INTERFACE ITF_CommunicationModul_1

METHOD Connect : BOOL
VAR_INPUT
END_VAR
END_METHOD

PROPERTY Connected : BOOL
GET
END_GET
END_PROPERTY

METHOD Disconnect : BOOL
VAR_INPUT
END_VAR
END_METHOD

METHOD ResetConnection : BOOL
VAR_INPUT
END_VAR
END_METHOD

END_INTERFACE

(* stored: Version 1.1.0.1, ProductVersion 3.1.4026.18
   Itf ITF_CommunicationModul_1: Id {8b7198f8-1e46-4b88-8db8-3a1ea1a87773}
   Method Connect: Id {83f24aef-d323-4734-92f2-2c83a095d25d}
   Property Connected: Id {fc1a5099-819f-456c-b0ef-9a99494a368f}
   Get Get: Id {98509eac-ca4d-438f-9ebc-9c88ffdd47d8}
   Method Disconnect: Id {b0eb8551-becc-4eec-a258-7ce9e2540525}
   Method ResetConnection: Id {c7dadd93-42f8-44ed-af9e-c44e6e8d20bc} *)
